PROGRAM prgLab08
VAR
	writePersistent:FB_WritePersistentData;
	error: BOOL;
	start: BOOL;
END_VAR
VAR PERSISTENT
	iPersistLocal:INT;
END_VAR

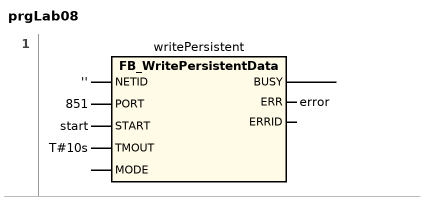
// NETWORK 1
writePersistent(NETID := '', PORT := 851, START := start, TMOUT := T#10s, ERR => error); // FB_WritePersistentData

END_PROGRAM

(* stored: Version 1.1.0.1, ProductVersion 3.1.4024.11
   POU prgLab08: Id {b1867b59-3131-45db-8c10-bcf88efae025}, SpecialFunc None *)
